# EPICS substitutions: iocs/ur621/iocBoot/iocur621/substitutions/fb_epid.substitutions
# $Id$

file "$(OPTICS)/opticsApp/Db/fb_epid.db"
  {
    {
        P=ur621:epid1,
	IN=ur621:epid1:sim.VAL,
	OUT=ur621:epid1:sim.D,
	MODE=PID,
	CALC=A,
	PERMIT1="ur621:epid1:on.VAL",
	PERMIT2="",
	PERMIT3="",
	PERMIT4=""
    }
  }
